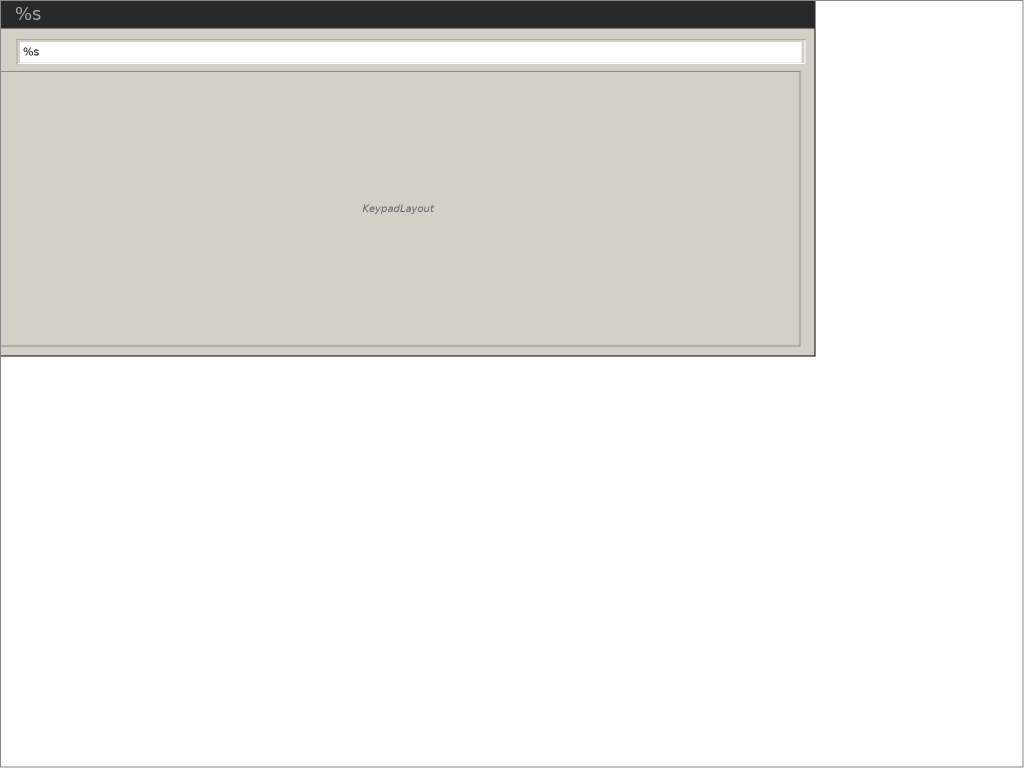
VISUALIZATION Keypad  // 1024x768
VAR_INPUT
	stVariableValue : STRING;
	stMin : STRING;
	stMax : STRING;
	wstTitle : WSTRING;
	flags : DWORD;
END_VAR
VAR
	bInit : BOOL;
	bShift : BOOL := TRUE;
	stMessage : STRING;
	stOutputValue : STRING;
	iCaretPosition	: INT;
	iSelectionStart	: INT;
	iSelectionEnd	: INT;
	xAllSelected	: BOOL;
END_VAR
    Rectangle (0,0 815x356)
    Polyline (17,64) (17,39) (805,39)
    Polyline (18,63) (805,63) (805,40)
    Textfield (20,42 781x20), "%s", text variable: stOutputValue
        p905179711: iCaretPosition
        p3815007873: iSelectionStart
        p1425650380: iSelectionEnd
        p3479897389: xAllSelected
    Rectangle (0,0 815x28), invisible if: VisuElems.g_VisualizationStyle.GetDINT('Dialog-UseHeaderColor', 0, 0) = 0
    Rectangle (12,4 793x20), "%s", text variable: gsPadTitle
    Frame (-3,71 803x275)
        shows KeypadLayout(stVariableValue := stVariableValue, bInit := bInit, bShift := bShift, stOutputValue := stOutputValue, iCaretPosition := iCaretPosition, iSelectionStart := iSelectionStart, iSelectionEnd := iSelectionEnd, flags := flags)
END_VISUALIZATION

(* stored: Version 1.1.0.1, ProductVersion 3.1.4024.2
   Visu Keypad: Id {a1635857-e90b-4bde-ba3e-416da4d089da} *)
